FUNCTION_BLOCK MoveSwitchToPosition
VAR_INPUT
END_VAR
VAR_OUTPUT
END_VAR
VAR
	moveAbs	: MC_MoveAbsolute;
	_axis : REFERENCE TO AXIS_REF;
	State: INT;
	_MoveSwitch : BOOL;
	_busy : BOOL;
	_error : BOOL;
	_done : BOOL;
END_VAR

CASE State OF
	0:
		IF _MoveSwitch THEN
			_done := FALSE;
			_error := FALSE;
			_busy := TRUE;
			moveAbs.Execute := TRUE;
			IF moveAbs.Busy THEN
				State := 10;
				_MoveSwitch := FALSE;
			END_IF
		END_IF
		
	10:
		IF NOT moveAbs.Busy THEN
			IF moveAbs.Done THEN
				_done := TRUE;
			ELSIF moveAbs.Error THEN
				_error := TRUE;
			END_IF
			_busy := FALSE;
			moveAbs.Execute := FALSE;
			State := 0;
		END_IF
END_CASE

moveAbs(Axis := _axis);

METHOD Abort : BOOL
moveAbs.Execute := FALSE;
moveAbs.Position := moveAbs.Velocity := 0;
_MoveSwitch := false;
_busy := false;
Abort := true;
State := 0;
END_METHOD

PROPERTY PUBLIC Acceleration : mc_lreal
GET
Acceleration := moveAbs.Acceleration;
END_GET
SET
moveAbs.Acceleration := Acceleration;
END_SET
END_PROPERTY

PROPERTY Busy : BOOL
GET
Busy := _busy;
END_GET
END_PROPERTY

PROPERTY PUBLIC Deceleration : mc_lreal
GET
Deceleration := moveAbs.Deceleration;
END_GET
SET
moveAbs.Deceleration := Deceleration;
END_SET
END_PROPERTY

PROPERTY Done : BOOL
GET
Done := _done;
END_GET
END_PROPERTY

PROPERTY Error : BOOL
GET
Error := _error;
END_GET
END_PROPERTY

METHOD FB_init : BOOL
VAR_INPUT
	bInitRetains : BOOL; // if TRUE, the retain variables are initialized (warm start / cold start)
	bInCopyCode : BOOL;  // if TRUE, the instance afterwards gets moved into the copy code (online change)
	axis : reference TO AXIS_REF;
END_VAR
_axis REF= axis;
END_METHOD

PROPERTY PUBLIC Jerk : mc_lreal
GET
Jerk := moveAbs.Jerk;
END_GET
SET
moveAbs.Jerk := Jerk;
END_SET
END_PROPERTY

METHOD MoveTo : BOOL
VAR_INPUT
	Position : MC_LREAL;
	Velocity : MC_LREAL;
END_VAR
moveAbs.Position := Position;
moveAbs.Velocity := Velocity;
_MoveSwitch := MoveTo := true;
END_METHOD

END_FUNCTION_BLOCK

(* stored: Version 1.1.0.1, ProductVersion 3.1.4024.11
   POU MoveSwitchToPosition: Id {c7eeeee5-3b61-4557-b5ce-9b78a6d29876}, SpecialFunc None
   Method Abort: Id {fce17614-0d2c-4f6c-a59d-598919ecd7bc}
   Property Acceleration: Id {ee03a772-233b-4093-9712-e60ef4c62467}
   Get Get: Id {cc971db7-f450-4332-bd5f-4bf4a49c8076}
   Set Set: Id {088acb42-6243-42a1-bef7-4367063fc3e3}
   Property Busy: Id {e6260c26-dd4a-4875-94a8-dbe321c9cf67}
   Get Get: Id {21af624d-322e-43a5-90ae-40b255f730fc}
   Property Deceleration: Id {9eb34121-a694-49aa-bead-7e740482330e}
   Get Get: Id {7bb899ac-4236-4501-ba6e-0e47f4aced93}
   Set Set: Id {75c4a9bd-c04c-4f88-84db-ed1910824505}
   Property Done: Id {8de0a85a-6316-4555-8b97-9f7d0cda87db}
   Get Get: Id {7518dba5-8b03-49de-a6c1-382e70601996}
   Property Error: Id {6bcf472f-6b47-43bb-b30f-ed40c368e7e3}
   Get Get: Id {567ad00c-542e-4928-a570-38631342e583}
   Method FB_init: Id {9ba40879-82be-499f-b7a0-91e6d6e7748a}
   Property Jerk: Id {34b2c07e-44a5-41d5-8ac6-37a9b7eb8cf3}
   Get Get: Id {00396a86-70c9-49a3-9e1d-d549b8ef933a}
   Set Set: Id {b9be6dc4-5427-4c77-84d5-c8637c0a22f1}
   Method MoveTo: Id {2d453548-6733-488b-87af-92ec1e6cf430} *)
